{attribute 'qualified_only'}
{attribute 'strict'}
TYPE eDeviceType :
(
	Unknown := 0,
	Primary := 1,
	Secondary := 2,
	Remote := 3
);
END_TYPE

(* stored: Version 1.1.0.1, ProductVersion 3.1.4024.15
   EnumerationTextList eDeviceType: Id {ca6f4410-18fe-4eb0-8172-b9186c7b13bb} *)
